TYPE DUT_8BIT :
STRUCT
	bData:BITARR8;
END_STRUCT
END_TYPE

(* stored: Version 1.1.0.1, ProductVersion 3.1.4024.11
   DUT DUT_8BIT: Id {aefa07c2-bcc3-4c12-82d7-108f713b9bfb} *)
